{attribute 'qualified_only'}
VAR_GLOBAL	
	bMidStationCam	: BOOL;
	bInfeedCam		: BOOL;
	bOutfeedCam		: BOOL;
	bRejectCam		: BOOL;
	
	
END_VAR

(* stored: Version 1.1.0.1
   GVL Trig: Id {171765cd-b3e1-44a6-b6ea-efc245c6aa1f} *)
